TYPE ST_System_BHKW_Parameter :
STRUCT
	AutoQuittierung			: BOOL;
	Zeit_Vorl				: TIME;
	Zeit_Nachl				: TIME;
END_STRUCT
END_TYPE

(* stored: Version 1.1.0.1, ProductVersion 3.1.4024.9
   DUT ST_System_BHKW_Parameter: Id {fded06a6-48f3-4a59-9566-1b9ac573cef9} *)
